(* CODESYS project CtaSysLeistungsventile_2.0.0.0.library
   Description: SYS Leistungventil Library der CTA
   Version: 2.0.0.0
   Title: CtaSysLeistungventile
   Author: SIS
   DocFormat: reStructuredText
   LanguageModelAttribute: qualified-access-only
   Placeholder: CtaSysLeistungventile
   CompiledLibraryCompatibilityVersion: CODESYS V3.5 SP16 Patch 3
   Company: CTA
   DefaultNamespace: CtaSysLeistungventile

Project tree, tasks and I/O mapping:
  libraries: Visu Utils, 4.5.0.0 (System); CtaAppBmk, 2.0.0.0 (CTA); CtaVisSymbols, 2.0.0.0 (CTA); VisuSymbols, 4.5.0.0 (System); CtaSysIO, 2.0.0.0 (CTA); CtaVisApps, 1.0.0.0 (CTA); CtaVisHelp, 1.0.0.0 (CTA); CtaVisUser, 1.0.0.0 (CTA)
  40 Visualizations/
    visualisation VIS_LEISTUNGSVENTILE_BASE
    visualisation VIS_LEISTUNGSVENTILE_BASE_ITF
    visualisation VIS_LEISTUNGSVENTILE_BASE_QUERRY
  00000000-0000-0000-0000-000000000000|D:\CoDeSys\LibrariesV3\trunk\Intern\CAA\CAA Template\3.4.0.0 draft\Placeholder.xml
  00000000-0000-0000-0000-000000000000|D:\CoDeSys\LibrariesV3\trunk\Intern\CAA\CAA Template\3.2.0.3 draft\Prefix.pdf
  00000000-0000-0000-0000-000000000000|D:\CoDeSys\LibrariesV3\trunk\Intern\CAA\CAA Template\3.5.2.0 draft\Placeholder.xml
  20 Structs/
  50 Images/
  10 Documenation/
    global variables VersionHistory
    global variables readMe
  21 Interface/
    interface ITF_LEISTUNGSVENTILE_BASE: proAcknowledge, proRelease, proVISU_DIA_NAME, proCR1, proCR2, proCR3, proCR4, proCAP, proITF_BMK_Verdichter
  11 Library Parameter/
  12 Konstanten/
  60 Textlisten/
    text list Error
    text list Info
    text list Warnung
  13 Globale Variablen/
  text list GlobalTextList
  5ce3da45-db07-42e7-a21c-a00fff4ed8f6|C:\Users\sis\Downloads\dip-switch.svg
  5ce3da45-db07-42e7-a21c-a00fff4ed8f6|C:\Users\sis\Downloads\lightning-bolt-circle.svg
  30 Program Organization Units/
    function block FB_LEISTUNGSVENTILE_BASE [ST]: proAcknowledge, proRelease, proVISU_DIA_NAME, proCAP, proCR1, proCR2, proCR3, proCR4, proITF_BMK_Verdichter
  5ce3da45-db07-42e7-a21c-a00fff4ed8f6|C:\Users\sis\Downloads\sine-wave.svg
  5ce3da45-db07-42e7-a21c-a00fff4ed8f6|C:\Users\sis\Downloads\eye.svg
  5ce3da45-db07-42e7-a21c-a00fff4ed8f6|C:\Users\sis\Downloads\lan.svg
*)

// 10 Documenation/VersionHistory
(* 

.. image:: ../../Images/CTA_Logo.jpg
   :align: right
   :width: 15% 

**Vorlage**   


============ =========== =========== ============================================
**Date**     **Version** **Author**  **Change**
------------ ----------- ----------- --------------------------------------------
04.03.2021   0.0.0.0     SIS         Vorlage erstellt

============ =========== =========== ============================================


*)
VAR_GLOBAL
    stInfo : STRING:= '0.0.0.0, Vorlage, CTA';
END_VAR

// 10 Documenation/readMe
(*

**ReadMe**
 
|	**Empfehlung**
|
|	Dokumentrieren Sie die Library für eine nachhaltige Entwicklung
|     
| *Beispiel*
| 
| Dies ist die Vorlage Library der CTA. Erstellen Sie ihre Library anhand dieser Vorlage.
*)

VAR_GLOBAL
    xReadMeDone              :   BOOL;
END_VAR

// 30 Program Organization Units/FB_LEISTUNGSVENTILE_BASE
FUNCTION_BLOCK FB_LEISTUNGSVENTILE_BASE IMPLEMENTS ITF_LEISTUNGSVENTILE_BASE

VAR
	// RELEASE
	xRelease        	:   BOOL;
	
    // RÜCKMELDUNG
	xAcknowledge    	:   BOOL;
	
   	// DIALOGNAME
	stVisuDiaName		:	STRING;
	
	// ITF AUF VENTILE
	ITF_xCR1_ON			:	CtaSysIO.ITF_IO;
	ITF_xCR2_ON			:	CtaSysIO.ITF_IO;
	ITF_xCR3_ON			:	CtaSysIO.ITF_IO;
	ITF_xCR4_ON			:	CtaSysIO.ITF_IO;	
	
	// VENTILE
	xCR1				:	BOOL;
	xCR2				:	BOOL;
	xCR3				:	BOOL;
	xCR4				:	BOOL;
	
	// KÄLTELEISTUNG
	iCAP				:	INT := 25;
	
	// BMK
	ITF_BMK				:	CtaAppBmk.ITF_BMK;
	
END_VAR

PROPERTY proAcknowledge : BOOL
GET
proAcknowledge := xAcknowledge;
END_GET
SET
xAcknowledge := proAcknowledge;
END_SET
END_PROPERTY

PROPERTY proRelease : BOOL
GET
proRelease := xRelease;
END_GET
SET
xRelease := proRelease;
END_SET
END_PROPERTY

PROPERTY proVISU_DIA_NAME : STRING
GET
proVISU_DIA_NAME := stVisuDiaName;
END_GET
END_PROPERTY

PROPERTY proCAP : INT
GET
proCAP	:= iCAP;
END_GET
END_PROPERTY

PROPERTY proCR1 : BOOL
GET
proCR1	:=	xCR1;
END_GET
END_PROPERTY

PROPERTY proCR2 : BOOL
GET
proCR2	:=	xCR2;
END_GET
END_PROPERTY

PROPERTY proCR3 : BOOL
GET
proCR3	:=	xCR3;
END_GET
END_PROPERTY

PROPERTY proCR4 : BOOL
GET
proCR4	:=	xCR4;
END_GET
END_PROPERTY

PROPERTY proITF_BMK_Verdichter : CtaAppBmk.ITF_BMK;
SET
ITF_BMK := proITF_BMK_Verdichter;
END_SET
END_PROPERTY

END_FUNCTION_BLOCK

// 21 Interface/ITF_LEISTUNGSVENTILE_BASE
INTERFACE ITF_LEISTUNGSVENTILE_BASE EXTENDS __System.IQueryInterface

PROPERTY proAcknowledge : BOOL
GET
END_GET
SET
END_SET
END_PROPERTY

PROPERTY proRelease : BOOL
GET
END_GET
SET
END_SET
END_PROPERTY

PROPERTY proVISU_DIA_NAME : STRING
GET
END_GET
END_PROPERTY

PROPERTY proCR1 : BOOL
GET
END_GET
END_PROPERTY

PROPERTY proCR2 : BOOL
GET
END_GET
END_PROPERTY

PROPERTY proCR3 : BOOL
GET
END_GET
END_PROPERTY

PROPERTY proCR4 : BOOL
GET
END_GET
END_PROPERTY

PROPERTY proCAP : INT
GET
END_GET
END_PROPERTY

PROPERTY proITF_BMK_Verdichter : CtaAppBmk.ITF_BMK;
SET
END_SET
END_PROPERTY

END_INTERFACE

// 40 Visualizations/VIS_LEISTUNGSVENTILE_BASE
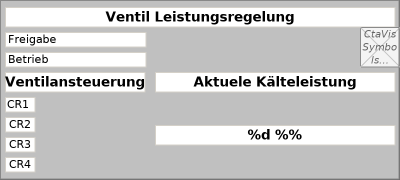
VISUALIZATION VIS_LEISTUNGSVENTILE_BASE  // 400x180
VAR_INPUT
	ITF_LEISTUNGSVENTILE_BASEIn   :   ITF_LEISTUNGSVENTILE_BASE;
END_VAR
    Frame (0,0 400x180), invisible if: NOT __QUERYINTERFACE(ITF_LEISTUNGSVENTILE_BASEIn,ITF_LEISTUNGSVENTILE_BASEIn)
        shows VIS_LEISTUNGSVENTILE_BASE_QUERRY(ITF_LEISTUNGSVENTILE_BASEIn := ITF_LEISTUNGSVENTILE_BASEIn)
END_VISUALIZATION

// 40 Visualizations/VIS_LEISTUNGSVENTILE_BASE_ITF
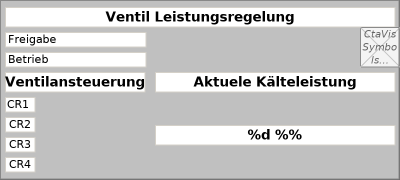
VISUALIZATION VIS_LEISTUNGSVENTILE_BASE_ITF  // 400x180
VAR_INPUT
	ITF_LEISTUNGSVENTILE_BASEIn   :   ITF_LEISTUNGSVENTILE_BASE;
END_VAR
VAR
    fbDialog    	:   VU.FbOpenDialogExtended;
END_VAR
    Rectangle (0,0 400x180)
    Textfield (5,7 390x20), "Ventil Leistungsregelung"
    Image (360,27 40x40), invisible if: ITF_LEISTUNGSVENTILE_BASEIn.proVISU_DIA_NAME = '', input disabled if: ITF_LEISTUNGSVENTILE_BASEIn.proVISU_DIA_NAME = '', image: CtaVisSymbols.ImagePool.gear
        OnMouseClick: execute {
            fbDialog(itfClientFilter            := VU.Globals.CurrentClient,
                     xExecute                   := FALSE,
                     sDialogName                := ITF_LEISTUNGSVENTILE_BASEIn.proVISU_DIA_NAME,
                     pbyDialogInterfaceData     := ADR(ITF_LEISTUNGSVENTILE_BASEIn),
                     udiDialogInterfaceDataSize := SIZEOF(ITF_LEISTUNGSVENTILE_BASEIn));
            fbDialog(itfClientFilter            := VU.Globals.CurrentClient,
                     xExecute                   := TRUE,
                     sDialogName                := ITF_LEISTUNGSVENTILE_BASEIn.proVISU_DIA_NAME,
                     pbyDialogInterfaceData     := ADR(ITF_LEISTUNGSVENTILE_BASEIn),
                     udiDialogInterfaceDataSize := SIZEOF(ITF_LEISTUNGSVENTILE_BASEIn));
        }
    Textfield (5,32 141x15), "Freigabe", colour toggle: ITF_LEISTUNGSVENTILE_BASEIn.proRelease
    Textfield (5,52 141x15), "Betrieb", colour toggle: ITF_LEISTUNGSVENTILE_BASEIn.proAcknowledge
    Textfield (5,72 140x20), "Ventilansteuerung"
    Textfield (5,97 30x15), "CR1", colour toggle: ITF_LEISTUNGSVENTILE_BASEIn.proCR1
    Textfield (5,117 30x15), "CR2", colour toggle: ITF_LEISTUNGSVENTILE_BASEIn.proCR2
    Textfield (5,137 30x15), "CR3", colour toggle: ITF_LEISTUNGSVENTILE_BASEIn.proCR3
    Textfield (5,157 30x15), "CR4", colour toggle: ITF_LEISTUNGSVENTILE_BASEIn.proCR4
    Textfield (155,72 240x20), "Aktuele Kälteleistung"
    Textfield (155,125 240x20), "%d %%", text variable: ITF_LEISTUNGSVENTILE_BASEIn.proCAP
END_VISUALIZATION

// 40 Visualizations/VIS_LEISTUNGSVENTILE_BASE_QUERRY
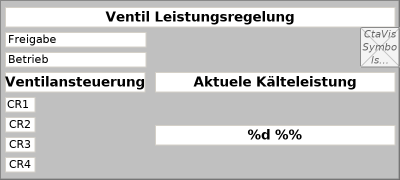
VISUALIZATION VIS_LEISTUNGSVENTILE_BASE_QUERRY  // 400x180
VAR_INPUT
	ITF_LEISTUNGSVENTILE_BASEIn   :   ITF_LEISTUNGSVENTILE_BASE;
END_VAR
    Frame (0,0 400x180), invisible if: NOT __QUERYINTERFACE(ITF_LEISTUNGSVENTILE_BASEIn,ITF_LEISTUNGSVENTILE_BASEIn)
        shows VIS_LEISTUNGSVENTILE_BASE_ITF(ITF_LEISTUNGSVENTILE_BASEIn := ITF_LEISTUNGSVENTILE_BASEIn)
END_VISUALIZATION

(* text list Error (id | default | de | en | fr | it)
  0 | keine Meldung Anstehend | Keine Meldung Anstehend | No message pending | Aucun message en attente | Nessun messaggio in sospeso
  1 | keine Betriebsrückmeldung | Keine Betriebsrückmeldung | No operational feedback | Aucune rétroaction opérationnelle | Nessun feedback operativo
  2 | Alarmkontakt Anstehend | Alarmkontakt Anstehend | Error contact pending | Contact d'alarme en attente | Contatto di allarme in sospeso
  3 | Leitungsschutzschalter ausfall | Leitungsschutzschalter ausfall | Circuit breaker failure | Défaillance du disjoncteur | Guasto dell'interruttore
  4 | Motorschutzschalter ausfall | Motorschutzschalter ausfall | Motor protection switch failure | Défaillance de l'interrupteur de protection du moteur | Guasto al salvamotore
  5 | Konfigurationsfehler speichern fehlgeschlagen reboot | Konfigurationsfehler speichern fehlgeschlagen reboot | Failed to save configuration error reboot | Impossible d'enregistrer l'erreur de configuration reboot | Impossibile salvare l'errore di configurazione reboot
   |  |  |  |  |  *)

(* text list Info (id | default | de | en | fr | it)
  0 | keine Meldung Anstehend | keine Meldung Anstehend | no message pending | aucun message en attente | nessun messaggio in sospeso
   |  |  |  |  |  *)

(* text list Warnung (id | default | de | en | fr | it)
  0 | Keine Meldung Anstehend | Keine Meldung Anstehend | No message pending | Aucun message en attente | Nessun messaggio in sospeso
  4 | Wahlschalter Hand, Ein | Wahlschalter Hand, Ein | Selector switch hand on | Commutateur de sélection a main, Allumé | Selettore a mano, acceso
  3 | Wahlschalter Hand, Aus | Wahlschalter Hand, Aus | Selector switch hand off | Commutateur de sélection a main, Éteint | Selettore a mano, spento
  2 | Revisionsschalter Ausgeschalten | Revisionsschalter Ausgeschalten | Revision switch off | Commutateur révision Désactiver | Interruttore di revisione disattivato
  1 | Sicherheits Stopp | Sicherheits Stopp | Safety stop | Arrêt de sécurité | Sosta di sicurezza
  5 | Handmodul aktiv | Handmodul aktiv | Hand module active | Module manuel actif | Modulo manuale attivo
   |  |  |  |  |  *)
